GLOBALCONSTANTS wordconst (* Global constants *)
  (* Standard: 61499-1 *)
  (* Version 1.0, 2024-02-22, franz *)
  VAR_GLOBAL CONSTANT
    DWORD_WORD_ZZ : DWORD := 16#0000_0000; (* ZERO Constant *)
    SHIFT_WORD_00 : SINT := 0; (* shift 0 bits *)
    DWORD_WORD_00 : DWORD := 16#0000_FFFF; (* LSB_Byte Constant *)
    SHIFT_WORD_01 : SINT := 16; (* shift 16 bits *)
    DWORD_WORD_01 : DWORD := 16#FFFF_0000; (* MSB_Byte Constant *)
  END_VAR
END_GLOBALCONSTANTS
